FUNCTION_BLOCK Motion_Control IMPLEMENTS ITF_MotionControl
VAR_INPUT
	HMI_MODE : BOOL;
END_VAR
VAR_OUTPUT
END_VAR
VAR
	AXIS_Object 	: POINTER TO Motion_Object;
	HmiToPlc		: POINTER TO Motion_HmiToPlc;
	PlcToHmi		: POINTER TO Motion_PlcToHmi;
	AXIS_COUNT		: INT := 0;
	HomeToNegative	: BOOL := TRUE;
	{attribute 'hide'}
	i				: INT;
	{attribute 'hide'}
	ptrPlcToHmi		: POINTER TO Motion_PlcToHmi;
	{attribute 'hide'}
	ptrHmiToPlc		: POINTER TO Motion_HmiToPlc;
	{attribute 'hide'}
	ptrAxisObj		: POINTER TO Motion_Object;
END_VAR

;

PROPERTY HmiToPlc_Address : POINTER TO Motion_HmiToPlc
SET
HmiToPlc := HmiToPlc_Address;
END_SET
END_PROPERTY

ACTION ACT_On:
On(i, HmiToPlc[i].ON_FW, HmiToPlc[i].ON_BW, HmiToPlc[i].CONTROLLER_OVERRIDE);
END_ACTION

PROPERTY PUBLIC InvertHomeDirection : BOOL
GET
InvertHomeDirection := HomeToNegative;
END_GET
SET
HomeToNegative := InvertHomeDirection;
END_SET
END_PROPERTY

METHOD PUBLIC Servo_isSoftLimitEnabled : ServoMotion_FunctionResult
VAR_INPUT
	INDEX 		: INT;
	OUTPUT 		: POINTER TO BOOL;
	POSITIVE	: BOOL; (*Targets the positive limit if true*)
END_VAR
VAR
	PARAMETER 	: MC_AxisParameter;
	BUFFER 		: BOOL;
END_VAR
IF INDEX > AXIS_COUNT OR INDEX < 1 THEN 
	Servo_isSoftLimitEnabled := Motion_FunctionResult.MOTION_UNKNOWN_AXIS;
ELSE
	IF POSITIVE THEN
		PARAMETER := MC_AxisParameter.EnableLimitPos;
	ELSE
		PARAMETER := MC_AxisParameter.EnableLimitNeg;
	END_IF
	fbRdParamBool[INDEX](
		Axis:= AXIS[INDEX].AXIS, 
		Enable:= TRUE, 
		ParameterNumber:= PARAMETER, 
		ReadMode:= ReadMode_Once, 
		Value=> BUFFER );
	IF fbRdParamBool[INDEX].Error THEN
		fbRdParamBool[INDEX](
			Axis:= AXIS[INDEX].AXIS, 
			Enable:= FALSE, 
			ParameterNumber:= PARAMETER, 
			ReadMode:= ReadMode_Once );
		Servo_isSoftLimitEnabled := Motion_FunctionResult.MOTION_ERROR;
	ELSIF NOT fbRdParamBool[INDEX].Busy THEN
		fbRdParamBool[INDEX](
			Axis:= AXIS[INDEX].AXIS, 
			Enable:= FALSE, 
			ParameterNumber:= PARAMETER, 
			ReadMode:= ReadMode_Once );
		OUTPUT^ := BUFFER;
		Servo_isSoftLimitEnabled := Motion_FunctionResult.MOTION_OK;
	ELSE
		Servo_isSoftLimitEnabled := Motion_FunctionResult.MOTION_BUSY;
	END_IF
END_IF
END_METHOD

METHOD PUBLIC Home : Motion_FunctionResult
VAR_INPUT
	INDEX : INT;
	//TO_NEGATIVE : BOOL;
END_VAR
VAR
	ptr_MotionObj : POINTER TO Motion_Object;
END_VAR
IF INDEX > AXIS_COUNT OR INDEX < 1 THEN 
	Home := Motion_FunctionResult.MOTION_UNKNOWN_AXIS;
ELSE
	ptr_MotionObj := Axis_Object + INT_TO_DWORD(INT_TO_UINT(INDEX -1) * SIZEOF(Motion_Object));
    Home := ptr_MotionObj^.Home(HomeToNegative);
END_IF
END_METHOD

METHOD PUBLIC Jog_Stop : Motion_FunctionResult
VAR_INPUT
	INDEX : INT;
END_VAR
VAR
	ptr_MotionObj : POINTER TO Motion_Object;
END_VAR
IF INDEX > AXIS_COUNT OR INDEX < 1 THEN 
	Jog_Stop := Motion_FunctionResult.MOTION_UNKNOWN_AXIS;
ELSE
	ptr_MotionObj := Axis_Object + INT_TO_DWORD(INT_TO_UINT(INDEX) * SIZEOF(Motion_Object));
    Jog_Stop := ptr_MotionObj^.Jog_Stop();
END_IF
END_METHOD

METHOD PUBLIC Off : Motion_FunctionResult
VAR_INPUT
	INDEX : INT;
END_VAR
VAR
	ptr_MotionObj : POINTER TO Motion_Object;
END_VAR
IF INDEX > AXIS_COUNT OR INDEX < 1 THEN 
	Off := Motion_FunctionResult.MOTION_UNKNOWN_AXIS;
ELSE
	ptr_MotionObj := Axis_Object + INT_TO_DWORD(INT_TO_UINT(INDEX - 1) * SIZEOF(Motion_Object));
    Off := ptr_MotionObj^.Off();
END_IF
END_METHOD

ACTION ACT_Halt:
CASE THIS^.Halt(i) OF 
Motion_FunctionResult.MOTION_UNKNOWN_AXIS:
	HmiToPlc^.HALT := FALSE;
Motion_FunctionResult.MOTION_ERROR:
	HmiToPlc^.HALT := FALSE;
Motion_FunctionResult.MOTION_OK:
	HmiToPlc^.HALT := FALSE;
Motion_FunctionResult.MOTION_COMMAND_ABORTED:
	HmiToPlc^.HALT := FALSE;
Motion_FunctionResult.MOTION_BUSY:
	;
END_CASE
END_ACTION

METHOD PUBLIC Servo_GetSoftLimit : ServoMotion_FunctionResult
VAR_INPUT
	INDEX 		: INT;
	OUTPUT 		: POINTER TO LREAL;
	POSITIVE	: BOOL; (*Targets the positive limit if true*)
END_VAR
VAR
	PARAMETER 	: MC_AxisParameter;
	BUFFER 		: LREAL;
END_VAR
IF INDEX > AXIS_COUNT OR INDEX < 1 THEN 
	Servo_GetSoftLimit := Motion_FunctionResult.MOTION_UNKNOWN_AXIS;
ELSE
	IF POSITIVE THEN
		PARAMETER := MC_AxisParameter.SWLimitPos;
	ELSE
		PARAMETER := MC_AxisParameter.SWLimitNeg;
	END_IF
	fbRdParam[INDEX](
		Axis:= AXIS[INDEX].AXIS, 
		Enable:= TRUE, 
		ParameterNumber:= PARAMETER, 
		ReadMode:= ReadMode_Once, 
		Value=> BUFFER);
	IF fbRdParam[INDEX].Error THEN
		fbRdParam[INDEX](
			Axis:= AXIS[INDEX].AXIS, 
			Enable:= FALSE, 
			ParameterNumber:= PARAMETER, 
			ReadMode:= ReadMode_Once );
		Servo_GetSoftLimit := Motion_FunctionResult.MOTION_ERROR;
	ELSIF NOT fbRdParam[INDEX].Busy THEN
		fbRdParam[INDEX](
			Axis:= AXIS[INDEX].AXIS, 
			Enable:= FALSE, 
			ParameterNumber:= PARAMETER, 
			ReadMode:= ReadMode_Once );
		OUTPUT^ := BUFFER;
		Servo_GetSoftLimit := Motion_FunctionResult.MOTION_OK;
	ELSE
		Servo_GetSoftLimit := Motion_FunctionResult.MOTION_BUSY;
	END_IF
END_IF
END_METHOD

METHOD PUBLIC Servo_EnableSoftLimit : ServoMotion_FunctionResult
VAR_INPUT
	INDEX 	: INT;
	POSITIVE: BOOL; (*Targets the positive limit if true*)
END_VAR
VAR
	PARAMETER 	: MC_AxisParameter;
	ENABLE 		: BOOL := TRUE;
END_VAR
IF INDEX > AXIS_COUNT OR INDEX < 1 THEN 
	Servo_EnableSoftLimit := Motion_FunctionResult.MOTION_UNKNOWN_AXIS;
ELSE
	IF POSITIVE THEN
		PARAMETER := MC_AxisParameter.EnableLimitPos;
	ELSE
		PARAMETER := MC_AxisParameter.EnableLimitNeg;
	END_IF
	fbSetParamBool[INDEX](
		Axis:= AXIS[INDEX].AXIS, 
		Execute:= TRUE, 
		ParameterNumber:= PARAMETER, 
		Value:= ENABLE );
	IF fbSetParamBool[INDEX].Error THEN
		fbSetParamBool[INDEX](
			Axis:= AXIS[INDEX].AXIS, 
			Execute:= FALSE, 
			ParameterNumber:= PARAMETER, 
			Value:= ENABLE);
		Servo_EnableSoftLimit := Motion_FunctionResult.MOTION_ERROR;
	ELSIF fbSetParamBool[INDEX].Done THEN
		fbSetParamBool[INDEX](
			Axis:= AXIS[INDEX].AXIS, 
			Execute:= FALSE, 
			ParameterNumber:= PARAMETER, 
			Value:= ENABLE );
		Servo_EnableSoftLimit := Motion_FunctionResult.MOTION_OK;
	ELSE
		Servo_EnableSoftLimit := ServoMotion_FunctionResult.MOTION_BUSY;
	END_IF
END_IF
END_METHOD

ACTION ACT_MoveToPosition:
CASE MoveToPosition(i,HmiToPlc[i].TARGET_POSITION,HmiToPlc[i].TARGET_VELOCITY,HmiToPlc[i].TARGET_ACCELERATION,HmiToPlc[i].TARGET_DECELERATION,HmiToPlc[i].TARGET_JERK) OF
Motion_FunctionResult.MOTION_UNKNOWN_AXIS:
	HmiToPlc^.MOVE_ABS := FALSE;
Motion_FunctionResult.MOTION_COMMAND_ABORTED: 
	HmiToPlc^.MOVE_ABS := FALSE;
Motion_FunctionResult.MOTION_ERROR:
	HmiToPlc^.MOVE_ABS := FALSE;
Motion_FunctionResult.MOTION_BUSY: 
	;
Motion_FunctionResult.MOTION_OK:
	HmiToPlc^.MOVE_ABS := FALSE;
END_CASE
END_ACTION

PROPERTY PUBLIC Count : INT
SET // PUBLIC
IF COUNT > 0 THEN
	AXIS_COUNT := COUNT;
END_IF
END_SET
GET
COUNT := AXIS_COUNT;
END_GET
END_PROPERTY

METHOD PUBLIC MoveToPosition : Motion_FunctionResult
VAR_INPUT
	INDEX 			: INT;
	POSITION		: LREAL;
	VELOCITY		: LREAL;
	ACCELERATION	: LREAL;
	DECELERATION	: LREAL;
	JERK			: LREAL;
END_VAR
VAR
	ptr_MotionObj : POINTER TO Motion_Object;
END_VAR
IF INDEX > AXIS_COUNT OR INDEX < 1 AND VELOCITY <= 0 THEN 
	MoveToPosition := Motion_FunctionResult.MOTION_UNKNOWN_AXIS;
ELSE
	ptr_MotionObj := Axis_Object + INT_TO_DWORD(INT_TO_UINT(INDEX - 1) * SIZEOF(Motion_Object));
    MoveToPosition := ptr_MotionObj^.MoveToPosition(POSITION,VELOCITY,ACCELERATION,DECELERATION,JERK);
END_IF
END_METHOD

PROPERTY PlcToHmi_Address : POINTER TO Motion_PlcToHmi
SET
PlcToHmi := PlcToHmi_Address;
END_SET
END_PROPERTY

METHOD PUBLIC Servo_SetSoftLimit : ServoMotion_FunctionResult
VAR_INPUT
	INDEX 	: INT;
	VALUE 	: LREAL;
	POSITIVE: BOOL; (*Targets the positive limit if true*)
END_VAR
VAR
	PARAMETER : MC_AxisParameter;
END_VAR
IF INDEX > AXIS_COUNT OR INDEX < 1 THEN 
	Servo_SetSoftLimit := Motion_FunctionResult.MOTION_UNKNOWN_AXIS;
ELSE
	IF POSITIVE THEN
		PARAMETER := MC_AxisParameter.SWLimitPos;
	ELSE
		PARAMETER := MC_AxisParameter.SWLimitNeg;
	END_IF
	fbSetParam[INDEX](
		Axis:= AXIS[INDEX].AXIS, 
		Execute:= TRUE, 
		ParameterNumber:= PARAMETER, 
		Value:= VALUE );
	IF fbSetParam[INDEX].Error THEN
		fbSetParam[INDEX](
			Axis:= AXIS[INDEX].AXIS, 
			Execute:= FALSE, 
			ParameterNumber:= PARAMETER, 
			Value:= VALUE );
		Servo_SetSoftLimit := Motion_FunctionResult.MOTION_ERROR;
	ELSIF fbSetParam[INDEX].Done THEN
		fbSetParam[INDEX](
			Axis:= AXIS[INDEX].AXIS, 
			Execute:= FALSE, 
			ParameterNumber:= PARAMETER, 
			Value:= VALUE );
		Servo_SetSoftLimit := Motion_FunctionResult.MOTION_OK;
	ELSE
		Servo_SetSoftLimit := Motion_FunctionResult.MOTION_BUSY;
	END_IF
END_IF
END_METHOD

ACTION ACT_Off:
Off(i);
END_ACTION

METHOD PUBLIC Halt : Motion_FunctionResult
VAR_INPUT
	INDEX : INT;
END_VAR
VAR
	ptr_MotionObj : POINTER TO Motion_Object;
END_VAR
IF INDEX > AXIS_COUNT OR INDEX < 1 THEN 
	Halt := Motion_FunctionResult.MOTION_UNKNOWN_AXIS;
ELSE
	ptr_MotionObj := Axis_Object + INT_TO_DWORD(INT_TO_UINT(INDEX -1) * SIZEOF(Motion_Object));
    Halt := ptr_MotionObj^.Halt();
END_IF
END_METHOD

ACTION ACT_MoveByDistance:
CASE THIS^.MoveByDistance(i,HmiToPlc[i].TARGET_POSITION,HmiToPlc[i].TARGET_VELOCITY,HmiToPlc[i].TARGET_ACCELERATION,HmiToPlc[i].TARGET_DECELERATION,HmiToPlc[i].TARGET_JERK) OF
Motion_FunctionResult.MOTION_UNKNOWN_AXIS:
	HmiToPlc^.MOVE_REL := FALSE;
Motion_FunctionResult.MOTION_COMMAND_ABORTED: 
	HmiToPlc^.MOVE_REL := FALSE;
Motion_FunctionResult.MOTION_ERROR:
	HmiToPlc^.MOVE_REL := FALSE;
Motion_FunctionResult.MOTION_BUSY: 
	;
Motion_FunctionResult.MOTION_OK:
	HmiToPlc^.MOVE_REL := FALSE;
END_CASE
END_ACTION

{attribute 'object_name' := 'HmiMode'}
METHOD HmiMode
FOR i := 1 TO AXIS_COUNT BY 1 DO
	ptrAxisObj := AXIS_Object + ((i-1) * SIZEOF(Motion_Object)); 
	ptrPlcToHmi := PlcToHmi + ((i-1) * SIZEOF(Motion_PlcToHmi)); 
	ptrHmiToPlc := HmiToPlc + ((i-1) * SIZEOF(Motion_HmiToPlc)); 
	ACT_UpdateStatus();
	IF HmiToPlc^.OFF THEN
		ACT_Off();
	ELSIF HmiToPlc^.ON THEN 
		ACT_On();
	END_IF
	IF HmiToPlc^.RESET THEN 
		ACT_Reset();
	END_IF
	IF NOT HmiToPlc^.JOG_MODE THEN 
		THIS^.Jog_Stop(i);
		IF HmiToPlc^.HALT THEN 
			ACT_Halt();
		ELSIF HmiToPlc^.MOVE_ABS THEN
			ACT_MoveToPosition();
		END_IF
		IF HmiToPlc^.MOVE_REL THEN
			ACT_MoveByDistance();
		END_IF
	ELSE
		ACT_Jog();
	END_IF
END_FOR
END_METHOD

METHOD PUBLIC Jog_Start : Motion_FunctionResult
VAR_INPUT
	INDEX		: INT;
	REVERSE		: BOOL := FALSE;
	FAST_MODE	: BOOL := FALSE;
END_VAR
VAR
	ptr_MotionObj : POINTER TO Motion_Object;
END_VAR
IF INDEX > AXIS_COUNT OR INDEX < 1 THEN 
	Jog_Start := Motion_FunctionResult.MOTION_UNKNOWN_AXIS;
ELSE
	ptr_MotionObj := Axis_Object + INT_TO_DWORD(INT_TO_UINT(INDEX -1) * SIZEOF(Motion_Object));
    Jog_Start := ptr_MotionObj^.Jog_Start(REVERSE,FAST_MODE);
END_IF
END_METHOD

ACTION ACT_Reset:
IF Reset(i) = Motion_FunctionResult.MOTION_OK THEN
	HmiToPlc^.RESET := FALSE;
END_IF
END_ACTION

METHOD PUBLIC MoveByDistance : Motion_FunctionResult
VAR_INPUT
	INDEX 			: INT;
	DISTANCE 		: LREAL;
	VELOCITY 		: LREAL;
	ACCELERATION 	: LREAL;
	DECELERATION 	: LREAL;
	JERK 			: LREAL;
END_VAR
VAR
	ptr_MotionObj : POINTER TO Motion_Object;
END_VAR
IF INDEX > AXIS_COUNT OR INDEX < 1 AND VELOCITY <= 0 THEN 
	MoveByDistance := Motion_FunctionResult.MOTION_UNKNOWN_AXIS;
ELSE
	ptr_MotionObj := Axis_Object + INT_TO_DWORD(INT_TO_UINT(INDEX - 1) * SIZEOF(Motion_Object));
    MoveByDistance := ptr_MotionObj^.MoveByDistance(DISTANCE,VELOCITY,ACCELERATION,DECELERATION,JERK);
END_IF
END_METHOD

ACTION ACT_Jog:
IF HmiToPlc^.JOG_FW_FAST THEN
	Jog_Start(i, FALSE, TRUE);
ELSIF HmiToPlc^.JOG_FW_SLOW THEN
	Jog_Start(i, FALSE, FALSE);
ELSIF HmiToPlc^.JOG_BW_FAST THEN
	Jog_Start(i, TRUE, TRUE);
ELSIF HmiToPlc^.JOG_BW_SLOW THEN
	Jog_Start(i, TRUE, FALSE);
ELSE
	Jog_Stop(i);
END_IF
END_ACTION

METHOD PUBLIC Servo_DisableSoftLimit : ServoMotion_FunctionResult
VAR_INPUT
	INDEX 	: INT;
	POSITIVE: BOOL; (*Targets the positive limit if true*)
END_VAR
VAR
	PARAMETER 	: MC_AxisParameter;
	ENABLE 		: BOOL := FALSE;
END_VAR
IF INDEX > AXIS_COUNT OR INDEX < 1 THEN 
	Servo_DisableSoftLimit := Motion_FunctionResult.MOTION_UNKNOWN_AXIS;
ELSE
	IF POSITIVE THEN
		PARAMETER := MC_AxisParameter.EnableLimitPos;
	ELSE
		PARAMETER := MC_AxisParameter.EnableLimitNeg;
	END_IF
	fbSetParamBool[INDEX](
		Axis:= AXIS[INDEX].AXIS, 
		Execute:= TRUE, 
		ParameterNumber:= PARAMETER, 
		Value:= ENABLE );
	IF fbSetParamBool[INDEX].Error THEN
		fbSetParamBool[INDEX](
			Axis:= AXIS[INDEX].AXIS, 
			Execute:= FALSE, 
			ParameterNumber:= PARAMETER, 
			Value:= ENABLE);
		Servo_DisableSoftLimit := Motion_FunctionResult.MOTION_ERROR;
	ELSIF fbSetParamBool[INDEX].Done THEN
		fbSetParamBool[INDEX](
			Axis:= AXIS[INDEX].AXIS, 
			Execute:= FALSE, 
			ParameterNumber:= PARAMETER, 
			Value:= ENABLE );
		Servo_DisableSoftLimit := Motion_FunctionResult.MOTION_OK;
	ELSE
		Servo_DisableSoftLimit := Motion_FunctionResult.MOTION_BUSY;
	END_IF
END_IF
END_METHOD

METHOD On : Motion_FunctionResult
VAR_INPUT
	INDEX : INT;
	ENABLE_FW 	: BOOL;
	ENABLE_BW	: BOOL;
	OVERRIDE	: LREAL;
END_VAR
VAR
	ptr_MotionObj : POINTER TO Motion_Object;
END_VAR
IF INDEX > AXIS_COUNT OR INDEX < 1 THEN 
	On := Motion_FunctionResult.MOTION_UNKNOWN_AXIS;
ELSE
	ptr_MotionObj := Axis_Object + INT_TO_DWORD(INT_TO_UINT(INDEX - 1) * SIZEOF(Motion_Object));
    On := ptr_MotionObj^.On(ENABLE_FW,ENABLE_BW,OVERRIDE);
END_IF
END_METHOD

METHOD PUBLIC Reset : Motion_FunctionResult
VAR_INPUT
	INDEX :INT;
END_VAR
VAR
	ptr_MotionObj : POINTER TO Motion_Object;
END_VAR
IF INDEX > AXIS_COUNT OR INDEX < 1 THEN 
	Reset := Motion_FunctionResult.MOTION_UNKNOWN_AXIS;
ELSE
	ptr_MotionObj := Axis_Object + INT_TO_DWORD(INT_TO_UINT(INDEX - 1) * SIZEOF(Motion_Object));
    Reset := ptr_MotionObj^.Reset();
END_IF
END_METHOD

ACTION ACT_UpdateStatus:
ptrPlcToHmi^ := ptrAxisObj^.ToHmi;
END_ACTION

PROPERTY AXIS : POINTER TO Motion_Object
SET
AXIS_Object := AXIS;
END_SET
END_PROPERTY

END_FUNCTION_BLOCK

(* stored: Version 1.1.0.1, ProductVersion 3.1.4018.2
   POU Motion_Control: Id {55b379f4-f721-4632-9623-aca35a4ff0b7}, SpecialFunc None
   Folder Methods: Id {17551b9c-2969-46ec-8e71-0b07d9c32552}
   Folder NewFolder1: Id {36c71718-3734-4842-86fa-60ef735692e9}
   Folder Properties: Id {705af329-ccbe-4f33-b4ad-e8be6087764d}
   Folder HMI Actions: Id {a81ee722-85c9-42c1-866f-016e6d583404}
   Property HmiToPlc_Address: Id {04fea5c3-fc2d-45ae-8f6b-8c737924b0a6}
   Set Set: Id {de52f853-b5b9-4953-848d-3b44041cbcb0}
   Action ACT_On: Id {055125fe-25ee-4a7a-b050-73eb03772677}
   Property InvertHomeDirection: Id {07561adb-093e-4829-8253-55deb4091056}
   Get Get: Id {900c518b-2835-4c5b-80c3-b13012845d2a}
   Set Set: Id {def61d6e-0d36-466d-a2fe-ef3bddca370b}
   Method Servo_isSoftLimitEnabled: Id {09f570f6-1156-4979-bc4b-e6dd698d14fd}
   Method Home: Id {177da0d7-0e75-4752-b88f-e867267c266c}
   Method Jog_Stop: Id {1f8fc547-a813-4b5f-93fa-9fae40058f6f}
   Method Off: Id {2b7678fb-5114-4046-a0d3-11070b4fbd98}
   Action ACT_Halt: Id {39e232ab-6ebc-4ec0-af7e-c3ba534cc123}
   Method Servo_GetSoftLimit: Id {3be7fdfb-1ff5-443e-be62-1460c56c5e7e}
   Method Servo_EnableSoftLimit: Id {3f19cd5c-fc50-48a0-8fee-377a9e7cddd3}
   Action ACT_MoveToPosition: Id {40847845-e28a-467f-8c2b-007d9c73cf9b}
   Property Count: Id {459cb5a1-6ab5-4653-9f1f-4943f3702408}
   Set Set: Id {6fb218ec-b5b3-46d4-afd0-a81260142c21}
   Get Get: Id {9be2d030-51e7-4e34-80b7-5636315565bf}
   Method MoveToPosition: Id {4b4bad53-575d-4566-847b-5df400e707ed}
   Property PlcToHmi_Address: Id {4f554a56-7ed4-4543-845a-974db235ce2c}
   Set Set: Id {eafc9df8-a304-4032-a888-ce6beb82e774}
   Method Servo_SetSoftLimit: Id {52585544-64ca-4d30-bcd5-f069244950d0}
   Action ACT_Off: Id {5bdb5604-b204-4401-92fa-0d357435d921}
   Method Halt: Id {6989ff12-21aa-479d-ad23-23232d5ecada}
   Action ACT_MoveByDistance: Id {7d58b39d-b312-4669-b3d1-c2d6a9066f91}
   Method HmiMode: Id {8518e72e-9841-4325-a812-a953b639b662}
   Method Jog_Start: Id {857d1325-691b-4e71-89f9-5cc1b73fa800}
   Action ACT_Reset: Id {a7a36296-4bd3-4c04-bfcc-ad271ca28fe6}
   Method MoveByDistance: Id {b7b49934-4930-4ea2-b772-a6e74f151dd6}
   Action ACT_Jog: Id {cc0383b4-9148-4bf0-9c5a-f7313178b54b}
   Method Servo_DisableSoftLimit: Id {d26238b2-c0d2-4136-b2aa-48e42e86b1b5}
   Method On: Id {d7c9e2a6-ab50-4fb9-bb77-ce0d39e7247b}
   Method Reset: Id {e126d8bd-3570-40c3-9468-28dd8d3340a4}
   Action ACT_UpdateStatus: Id {fc19d8f7-7aab-443d-a6b0-6c271a3d11f7}
   Property AXIS: Id {fd24b662-ad51-4b71-a65c-ddcefcbcb58f}
   Set Set: Id {202590d2-eb4f-4c08-b713-480e513dea0a} *)
